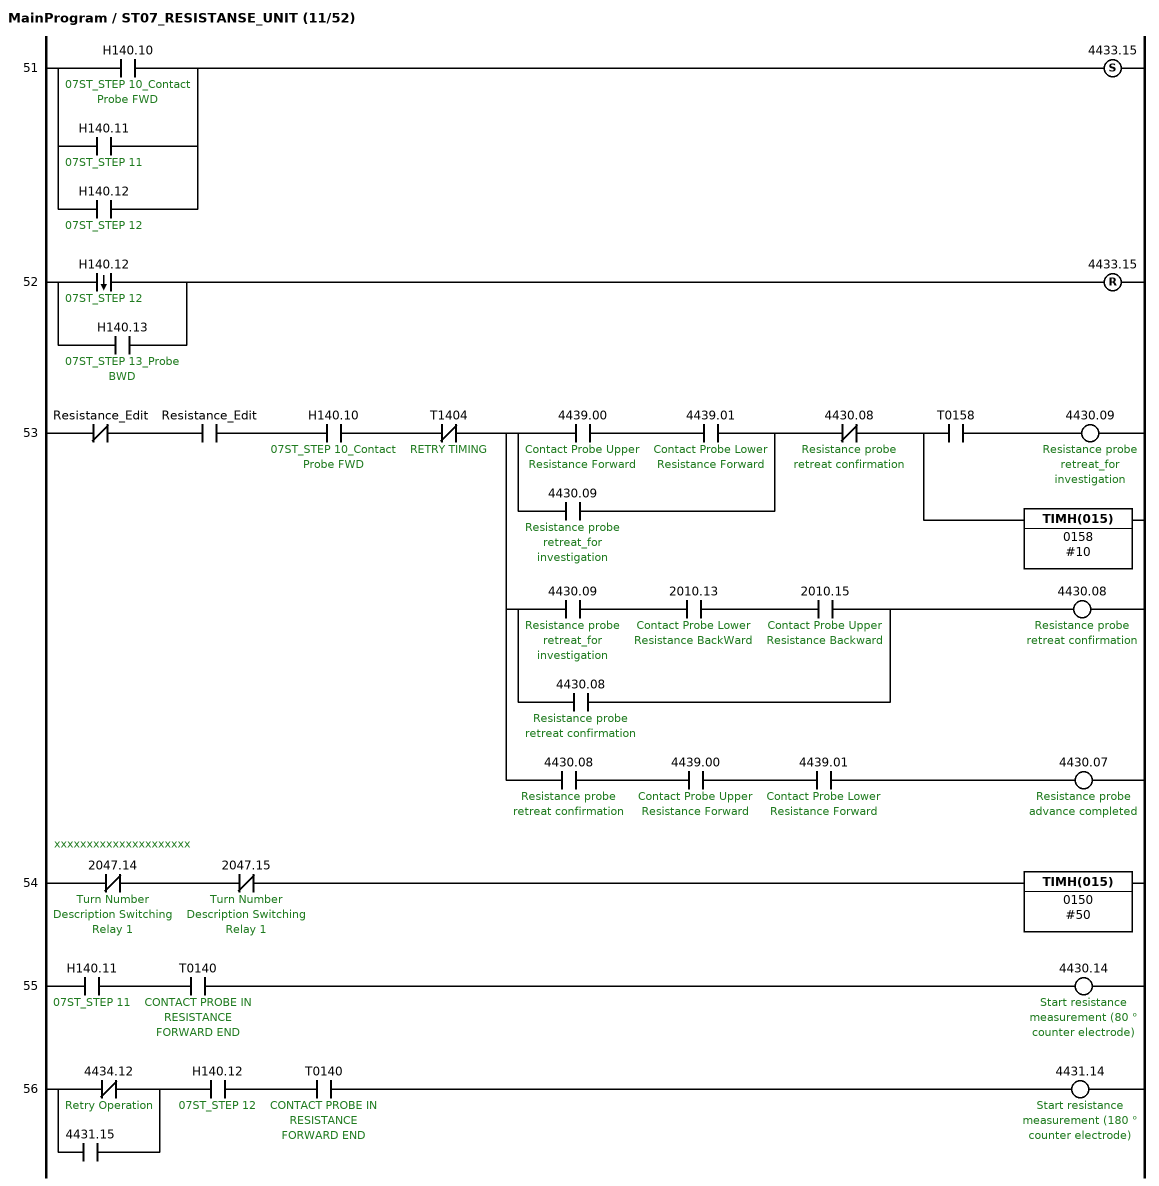
; [picture p384: MainProgram / ST07_RESISTANSE_UNIT, rungs 51-56]
; rung 51
LD H140.10  ; 07ST_STEP 10_Contact Probe FWD
OR H140.11  ; 07ST_STEP 11
OR H140.12  ; 07ST_STEP 12
SET 4433.15
; rung 52
%LD H140.12  ; 07ST_STEP 12
OR H140.13  ; 07ST_STEP 13_Probe BWD
RSET 4433.15
; rung 53
LDNOT Resistance_Edit
AND Resistance_Edit
AND H140.10  ; 07ST_STEP 10_Contact Probe FWD
ANDNOT T1404  ; RETRY TIMING
OUT TR0
LD 4439.00  ; Contact Probe Upper Resistance Forward
AND 4439.01  ; Contact Probe Lower Resistance Forward
OR 4430.09  ; Resistance probe retreat_for investigation
ANDLD
ANDNOT 4430.08  ; Resistance probe retreat confirmation
OUT TR1
AND T0158
OUT 4430.09  ; Resistance probe retreat_for investigation
LD TR1
TIMH(015) 0158 #10
LD TR0
LD 4430.09  ; Resistance probe retreat_for investigation
AND 2010.13  ; Contact Probe Lower Resistance BackWard
AND 2010.15  ; Contact Probe Upper Resistance Backward
OR 4430.08  ; Resistance probe retreat confirmation
ANDLD
OUT 4430.08  ; Resistance probe retreat confirmation
LD TR0
AND 4430.08  ; Resistance probe retreat confirmation
AND 4439.00  ; Contact Probe Upper Resistance Forward
AND 4439.01  ; Contact Probe Lower Resistance Forward
OUT 4430.07  ; Resistance probe advance completed
; rung 54: xxxxxxxxxxxxxxxxxxxxx
LDNOT 2047.14  ; Turn Number Description Switching Relay 1
ANDNOT 2047.15  ; Turn Number Description Switching Relay 1
TIMH(015) 0150 #50
; rung 55
LD H140.11  ; 07ST_STEP 11
AND T0140  ; CONTACT PROBE IN RESISTANCE FORWARD END
OUT 4430.14  ; Start resistance measurement (80 ° counter electrode)
; rung 56
LDNOT 4434.12  ; Retry Operation
OR 4431.15
AND H140.12  ; 07ST_STEP 12
AND T0140  ; CONTACT PROBE IN RESISTANCE FORWARD END
OUT 4431.14  ; Start resistance measurement (180 ° counter electrode)

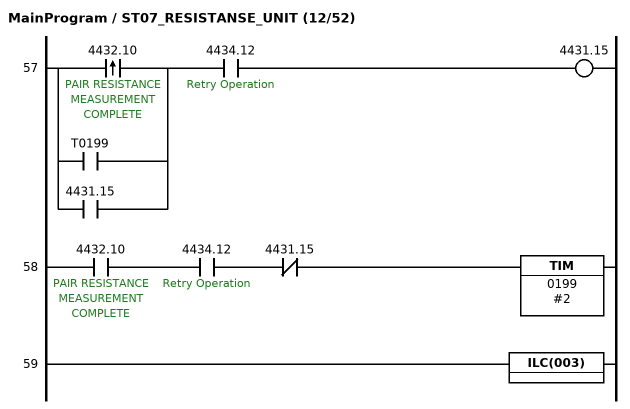
; rung 57
@LD 4432.10  ; PAIR RESISTANCE MEASUREMENT COMPLETE
OR T0199
OR 4431.15
AND 4434.12  ; Retry Operation
OUT 4431.15
; rung 58
LD 4432.10  ; PAIR RESISTANCE MEASUREMENT COMPLETE
AND 4434.12  ; Retry Operation
ANDNOT 4431.15
TIM 0199 #2
; rung 59
ILC(003)

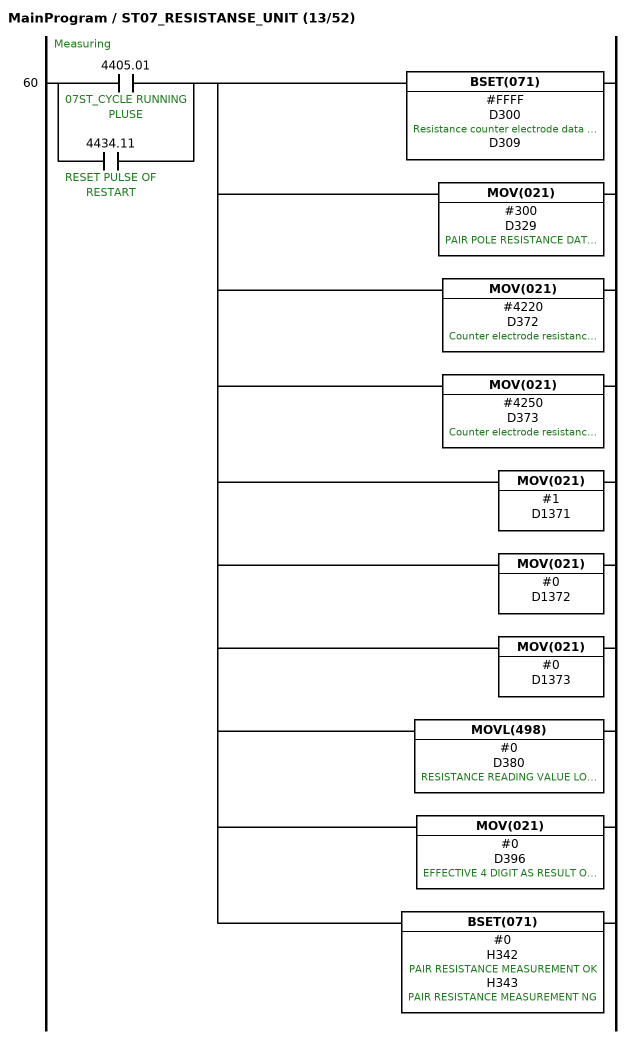
; rung 60: Measuring
LD 4405.01  ; 07ST_CYCLE RUNNING PLUSE
OR 4434.11  ; RESET PULSE OF RESTART
BSET(071) #FFFF D300 D309  ; Resistance counter electrode data 9 (80 ° counter electrode)
MOV(021) #300 D329  ; PAIR POLE RESISTANCE DATA INDIRECT SPECIFICATION
MOV(021) #4220 D372  ; Counter electrode resistance measurement indirect (80 °)
MOV(021) #4250 D373  ; Counter electrode resistance measurement indirect (80 °)
MOV(021) #1 D1371
MOV(021) #0 D1372
MOV(021) #0 D1373
MOVL(498) #0 D380  ; RESISTANCE READING VALUE LOW DIGIT
MOV(021) #0 D396  ; EFFECTIVE 4 DIGIT AS RESULT OF TEMPERATURE CORRECTION
BSET(071) #0 H342 H343  ; PAIR RESISTANCE MEASUREMENT OK, PAIR RESISTANCE MEASUREMENT NG

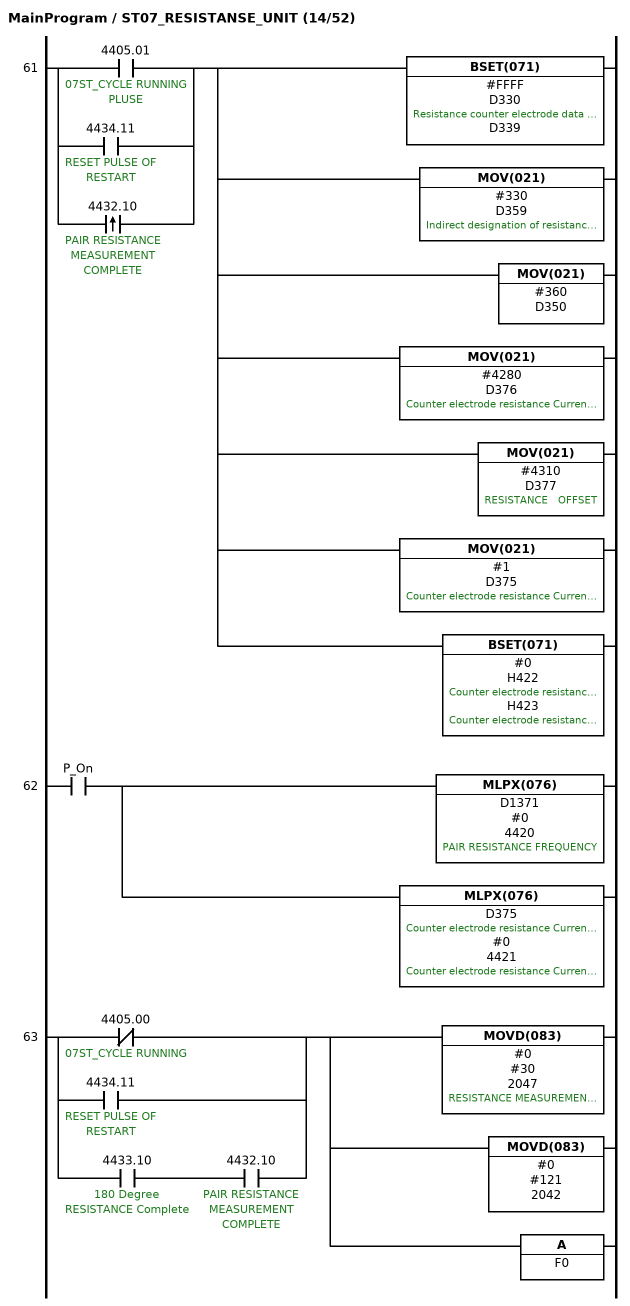
; rung 61
LD 4405.01  ; 07ST_CYCLE RUNNING PLUSE
OR 4434.11  ; RESET PULSE OF RESTART
@OR 4432.10  ; PAIR RESISTANCE MEASUREMENT COMPLETE
BSET(071) #FFFF D330 D339  ; Resistance counter electrode data 1 (180 ° counter electrode)
MOV(021) #330 D359  ; Indirect designation of resistance counter electrode data (180 °)
MOV(021) #360 D350
MOV(021) #4280 D376  ; Counter electrode resistance Current measurement count (180 °)
MOV(021) #4310 D377  ; RESISTANCE　OFFSET
MOV(021) #1 D375  ; Counter electrode resistance Current measurement count (180 °)
BSET(071) #0 H422 H423  ; Counter electrode resistance measurement OK (180 °), Counter electrode resistance measurement NG (180 °)
; rung 62
LD P_On
MLPX(076) D1371 #0 4420  ; PAIR RESISTANCE FREQUENCY
MLPX(076) D375 #0 4421  ; Counter electrode resistance Current measurement count (180 °)
; rung 63
LDNOT 4405.00  ; 07ST_CYCLE RUNNING
OR 4434.11  ; RESET PULSE OF RESTART
LD 4433.10  ; 180 Degree  RESISTANCE Complete
AND 4432.10  ; PAIR RESISTANCE MEASUREMENT COMPLETE
ORLD
MOVD(083) #0 #30 2047  ; RESISTANCE MEASUREMENT CHANGE RELAY
MOVD(083) #0 #121 2042
A  F0
// 

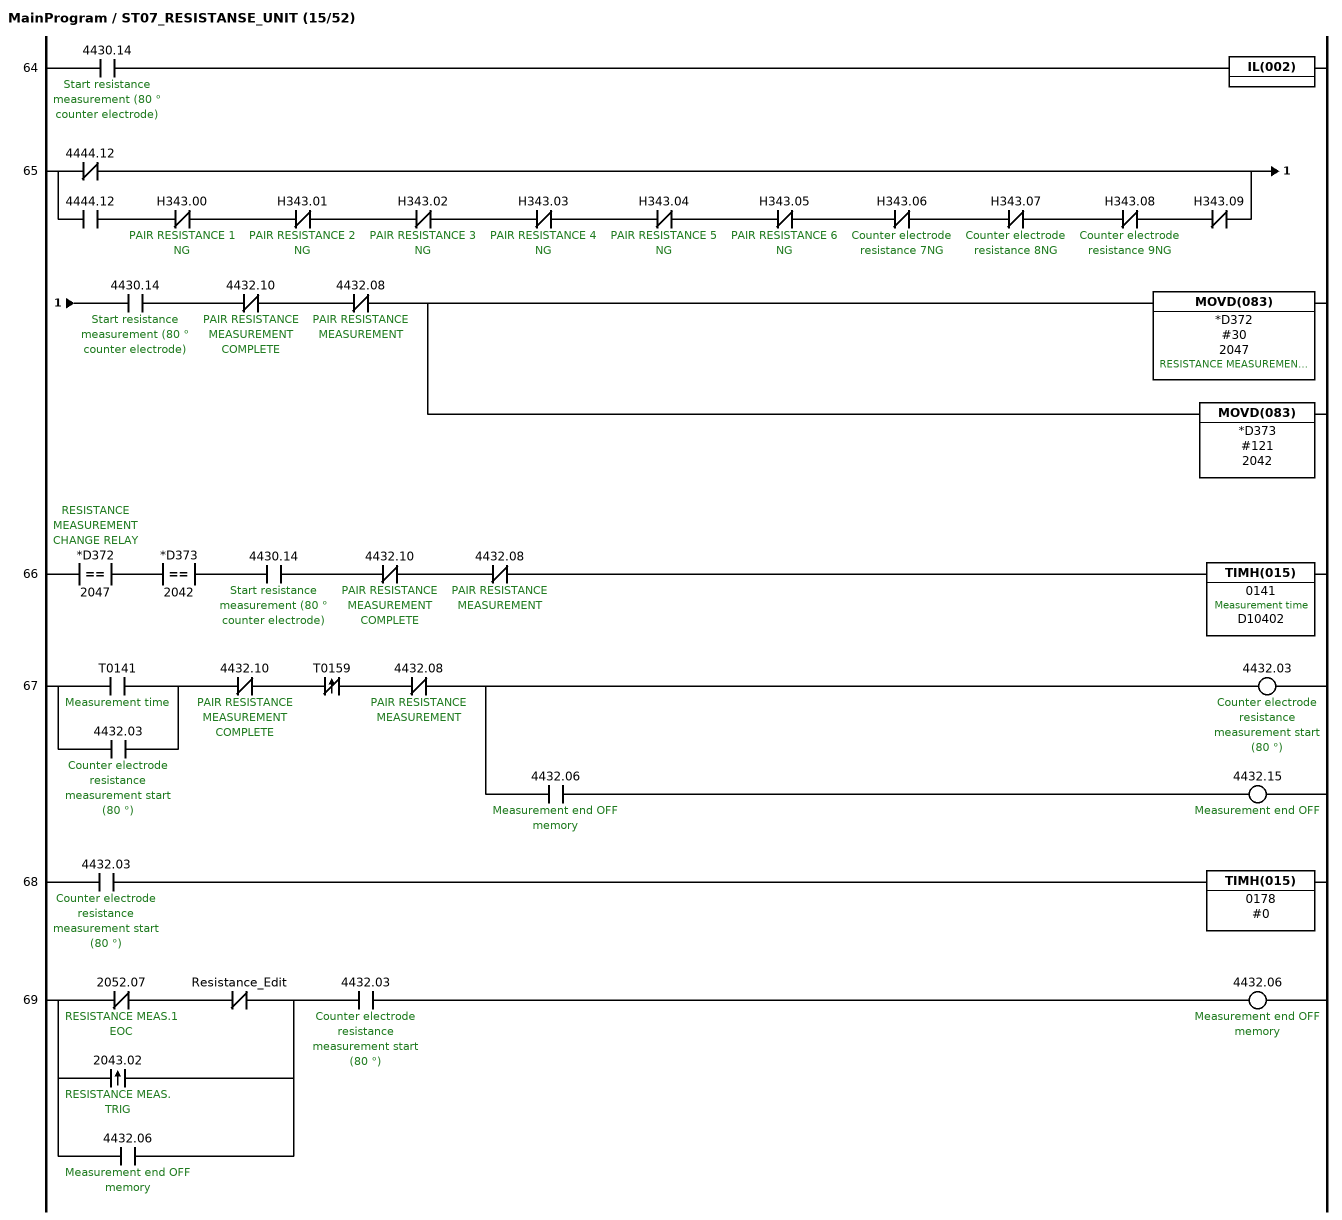
; rung 64
LD 4430.14  ; Start resistance measurement (80 ° counter electrode)
IL(002)
; rung 65
LDNOT 4444.12
LD 4444.12
ANDNOT H343.00  ; PAIR RESISTANCE 1 NG
ANDNOT H343.01  ; PAIR RESISTANCE 2 NG
ANDNOT H343.02  ; PAIR RESISTANCE 3 NG
ANDNOT H343.03  ; PAIR RESISTANCE 4 NG
ANDNOT H343.04  ; PAIR RESISTANCE 5 NG
ANDNOT H343.05  ; PAIR RESISTANCE 6 NG
ANDNOT H343.06  ; Counter electrode resistance 7NG
ANDNOT H343.07  ; Counter electrode resistance 8NG
ANDNOT H343.08  ; Counter electrode resistance 9NG
ANDNOT H343.09
ORLD
AND 4430.14  ; Start resistance measurement (80 ° counter electrode)
ANDNOT 4432.10  ; PAIR RESISTANCE MEASUREMENT COMPLETE
ANDNOT 4432.08  ; PAIR RESISTANCE MEASUREMENT
MOVD(083) *D372 #30 2047  ; RESISTANCE MEASUREMENT CHANGE RELAY
MOVD(083) *D373 #121 2042
; rung 66
LD=(300) *D372 2047  ; RESISTANCE MEASUREMENT CHANGE RELAY
AND=(300) *D373 2042
AND 4430.14  ; Start resistance measurement (80 ° counter electrode)
ANDNOT 4432.10  ; PAIR RESISTANCE MEASUREMENT COMPLETE
ANDNOT 4432.08  ; PAIR RESISTANCE MEASUREMENT
TIMH(015) 0141 D10402  ; Measurement time
; rung 67
LD T0141  ; Measurement time
OR 4432.03  ; Counter electrode resistance measurement start (80 °)
ANDNOT 4432.10  ; PAIR RESISTANCE MEASUREMENT COMPLETE
@ANDNOT T0159
ANDNOT 4432.08  ; PAIR RESISTANCE MEASUREMENT
OUT 4432.03  ; Counter electrode resistance measurement start (80 °)
AND 4432.06  ; Measurement end OFF memory
OUT 4432.15  ; Measurement end OFF
; rung 68
LD 4432.03  ; Counter electrode resistance measurement start (80 °)
TIMH(015) 0178 #0
; rung 69
LDNOT 2052.07  ; RESISTANCE MEAS.1 EOC
ANDNOT Resistance_Edit
@OR 2043.02  ; RESISTANCE MEAS. TRIG
OR 4432.06  ; Measurement end OFF memory
AND 4432.03  ; Counter electrode resistance measurement start (80 °)
OUT 4432.06  ; Measurement end OFF memory

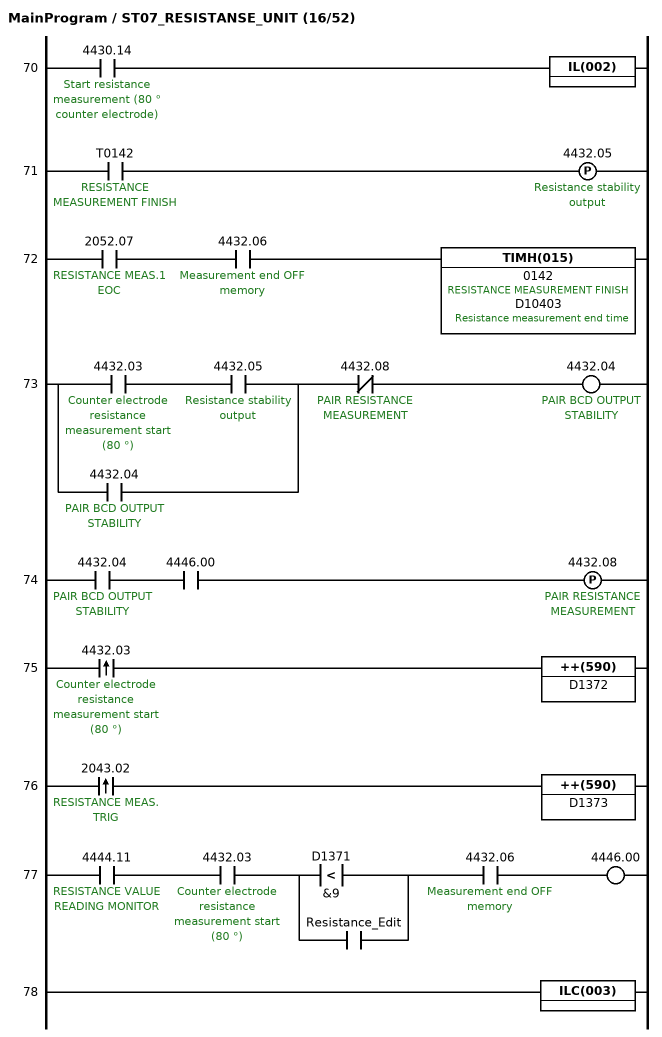
; rung 70
LD 4430.14  ; Start resistance measurement (80 ° counter electrode)
IL(002)
; rung 71
LD T0142  ; RESISTANCE MEASUREMENT FINISH
DIFU(013) 4432.05  ; Resistance stability output
; rung 72
LD 2052.07  ; RESISTANCE MEAS.1 EOC
AND 4432.06  ; Measurement end OFF memory
TIMH(015) 0142 D10403  ; Resistance measurement end time, RESISTANCE MEASUREMENT FINISH
; rung 73
LD 4432.03  ; Counter electrode resistance measurement start (80 °)
AND 4432.05  ; Resistance stability output
OR 4432.04  ; PAIR BCD OUTPUT STABILITY
ANDNOT 4432.08  ; PAIR RESISTANCE MEASUREMENT
OUT 4432.04  ; PAIR BCD OUTPUT STABILITY
; rung 74
LD 4432.04  ; PAIR BCD OUTPUT STABILITY
AND 4446.00
DIFU(013) 4432.08  ; PAIR RESISTANCE MEASUREMENT
; rung 75
@LD 4432.03  ; Counter electrode resistance measurement start (80 °)
++(590) D1372
; rung 76
@LD 2043.02  ; RESISTANCE MEAS. TRIG
++(590) D1373
; rung 77
LD 4444.11  ; RESISTANCE VALUE READING MONITOR
AND 4432.03  ; Counter electrode resistance measurement start (80 °)
LD<(310) D1371 &9
OR Resistance_Edit
ANDLD
AND 4432.06  ; Measurement end OFF memory
OUT 4446.00
; rung 78
ILC(003)

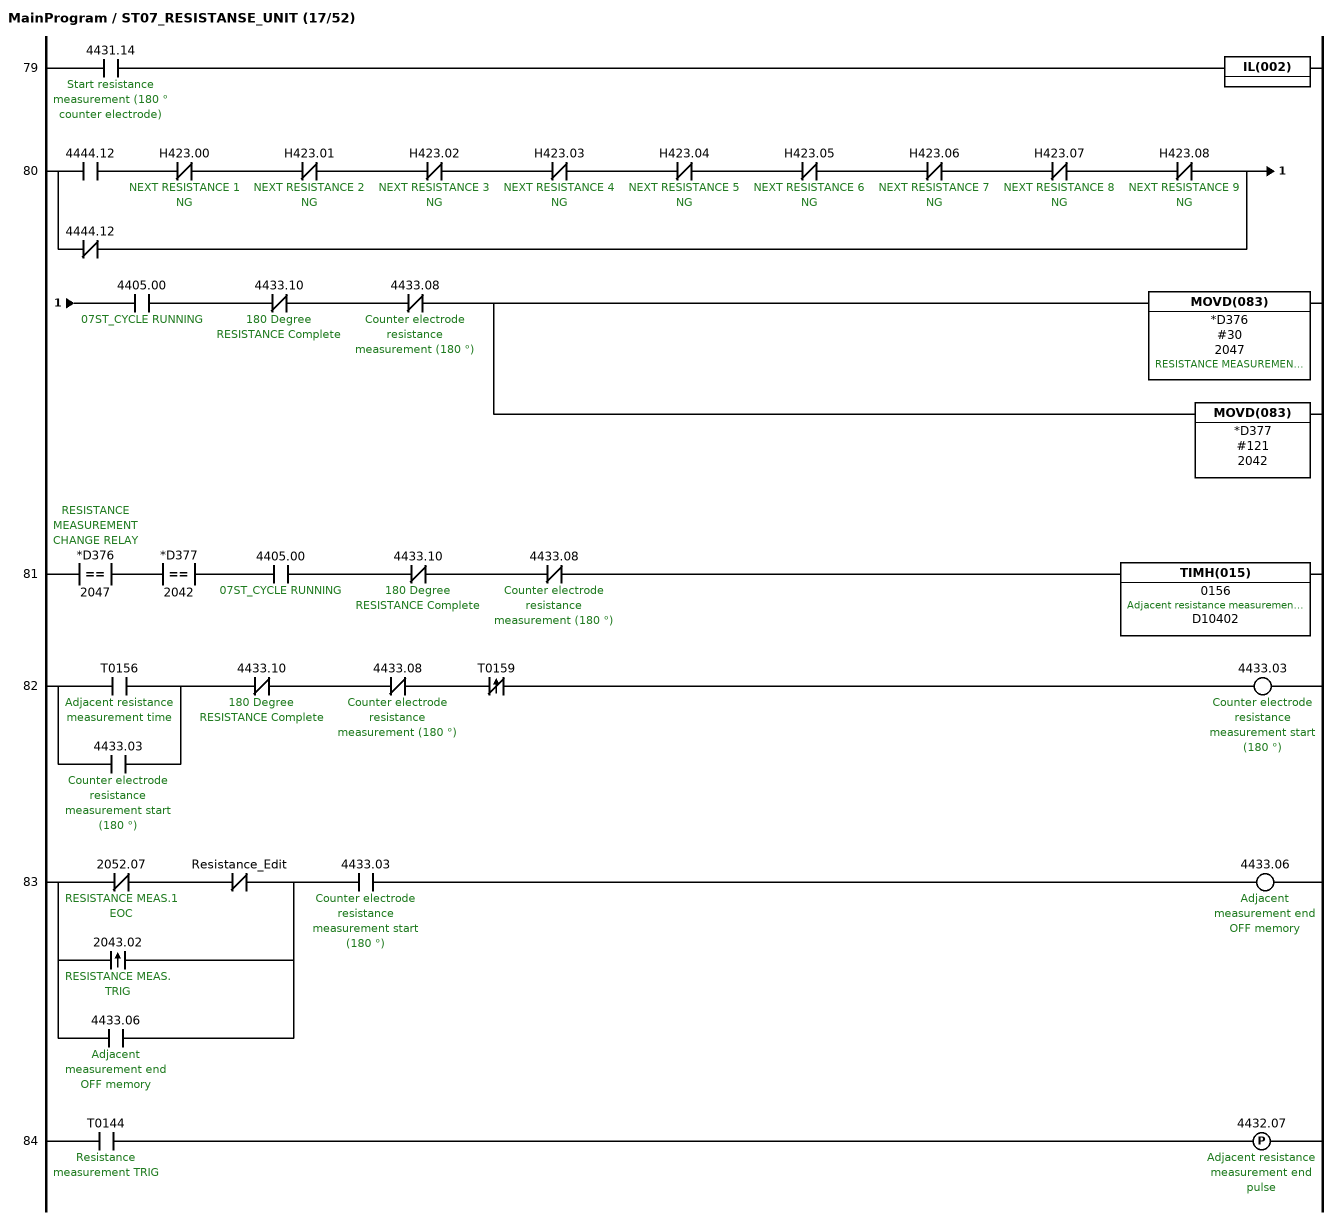
; rung 79
LD 4431.14  ; Start resistance measurement (180 ° counter electrode)
IL(002)
; rung 80
LD 4444.12
ANDNOT H423.00  ; NEXT RESISTANCE 1 NG
ANDNOT H423.01  ; NEXT RESISTANCE 2 NG
ANDNOT H423.02  ; NEXT RESISTANCE 3 NG
ANDNOT H423.03  ; NEXT RESISTANCE 4 NG
ANDNOT H423.04  ; NEXT RESISTANCE 5 NG
ANDNOT H423.05  ; NEXT RESISTANCE 6 NG
ANDNOT H423.06  ; NEXT RESISTANCE 7 NG
ANDNOT H423.07  ; NEXT RESISTANCE 8 NG
ANDNOT H423.08  ; NEXT RESISTANCE 9 NG
ORNOT 4444.12
AND 4405.00  ; 07ST_CYCLE RUNNING
ANDNOT 4433.10  ; 180 Degree  RESISTANCE Complete
ANDNOT 4433.08  ; Counter electrode resistance measurement (180 °)
MOVD(083) *D376 #30 2047  ; RESISTANCE MEASUREMENT CHANGE RELAY
MOVD(083) *D377 #121 2042
; rung 81
LD=(300) *D376 2047  ; RESISTANCE MEASUREMENT CHANGE RELAY
AND=(300) *D377 2042
AND 4405.00  ; 07ST_CYCLE RUNNING
ANDNOT 4433.10  ; 180 Degree  RESISTANCE Complete
ANDNOT 4433.08  ; Counter electrode resistance measurement (180 °)
TIMH(015) 0156 D10402  ; Adjacent resistance measurement time
; rung 82
LD T0156  ; Adjacent resistance measurement time
OR 4433.03  ; Counter electrode resistance measurement start (180 °)
ANDNOT 4433.10  ; 180 Degree  RESISTANCE Complete
ANDNOT 4433.08  ; Counter electrode resistance measurement (180 °)
@ANDNOT T0159
OUT 4433.03  ; Counter electrode resistance measurement start (180 °)
; rung 83
LDNOT 2052.07  ; RESISTANCE MEAS.1 EOC
ANDNOT Resistance_Edit
@OR 2043.02  ; RESISTANCE MEAS. TRIG
OR 4433.06  ; Adjacent measurement end OFF memory
AND 4433.03  ; Counter electrode resistance measurement start (180 °)
OUT 4433.06  ; Adjacent measurement end OFF memory
; rung 84
LD T0144  ; Resistance measurement TRIG
DIFU(013) 4432.07  ; Adjacent resistance measurement end pulse

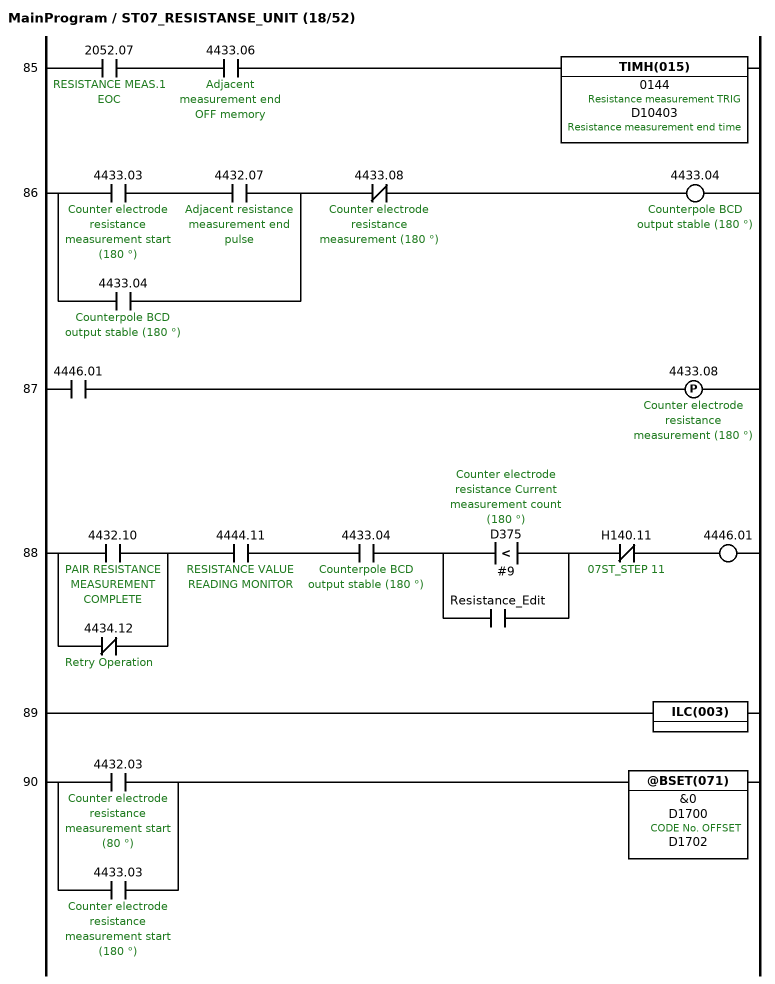
; rung 85
LD 2052.07  ; RESISTANCE MEAS.1 EOC
AND 4433.06  ; Adjacent measurement end OFF memory
TIMH(015) 0144 D10403  ; Resistance measurement end time, Resistance measurement TRIG
; rung 86
LD 4433.03  ; Counter electrode resistance measurement start (180 °)
AND 4432.07  ; Adjacent resistance measurement end pulse
OR 4433.04  ; Counterpole BCD output stable (180 °)
ANDNOT 4433.08  ; Counter electrode resistance measurement (180 °)
OUT 4433.04  ; Counterpole BCD output stable (180 °)
; rung 87
LD 4446.01
DIFU(013) 4433.08  ; Counter electrode resistance measurement (180 °)
; rung 88
LD 4432.10  ; PAIR RESISTANCE MEASUREMENT COMPLETE
ORNOT 4434.12  ; Retry Operation
AND 4444.11  ; RESISTANCE VALUE READING MONITOR
AND 4433.04  ; Counterpole BCD output stable (180 °)
LD<(310) D375 #9  ; Counter electrode resistance Current measurement count (180 °)
OR Resistance_Edit
ANDLD
ANDNOT H140.11  ; 07ST_STEP 11
OUT 4446.01
; rung 89
ILC(003)
; rung 90
LD 4432.03  ; Counter electrode resistance measurement start (80 °)
OR 4433.03  ; Counter electrode resistance measurement start (180 °)
@BSET(071) &0 D1700 D1702  ; CODE No. OFFSET

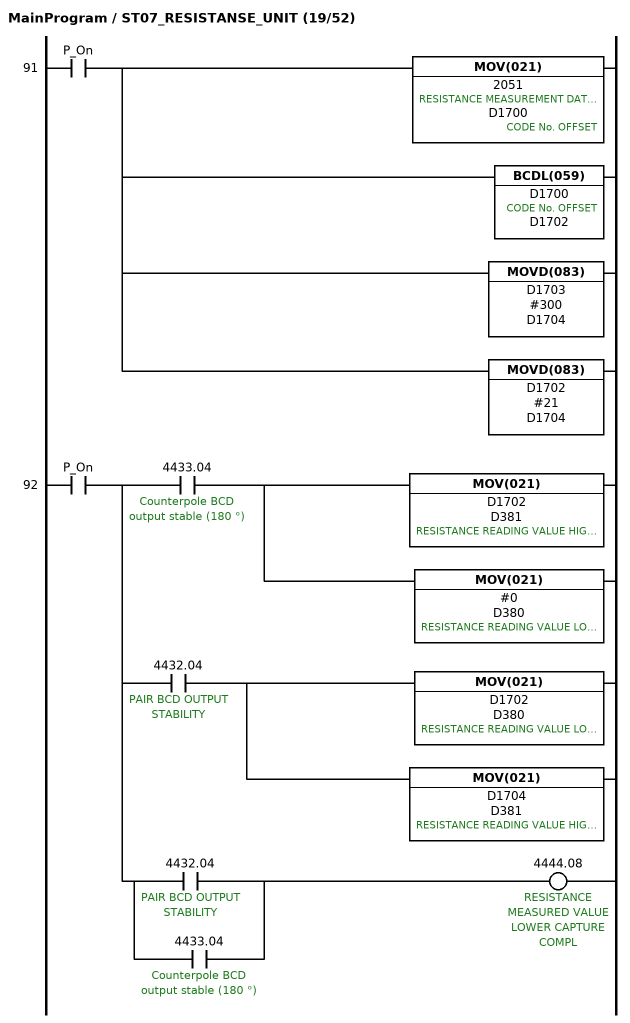
; rung 91
LD P_On
MOV(021) 2051 D1700  ; RESISTANCE MEASUREMENT DATA BCD, CODE No. OFFSET
BCDL(059) D1700 D1702  ; CODE No. OFFSET
MOVD(083) D1703 #300 D1704
MOVD(083) D1702 #21 D1704
; rung 92
LD P_On
OUT TR0
AND 4433.04  ; Counterpole BCD output stable (180 °)
MOV(021) D1702 D381  ; RESISTANCE READING VALUE HIGH DIGIT
MOV(021) #0 D380  ; RESISTANCE READING VALUE LOW DIGIT
LD TR0
AND 4432.04  ; PAIR BCD OUTPUT STABILITY
MOV(021) D1702 D380  ; RESISTANCE READING VALUE LOW DIGIT
MOV(021) D1704 D381  ; RESISTANCE READING VALUE HIGH DIGIT
LD TR0
LD 4432.04  ; PAIR BCD OUTPUT STABILITY
OR 4433.04  ; Counterpole BCD output stable (180 °)
ANDLD
OUT 4444.08  ; RESISTANCE MEASURED VALUE LOWER CAPTURE COMPL

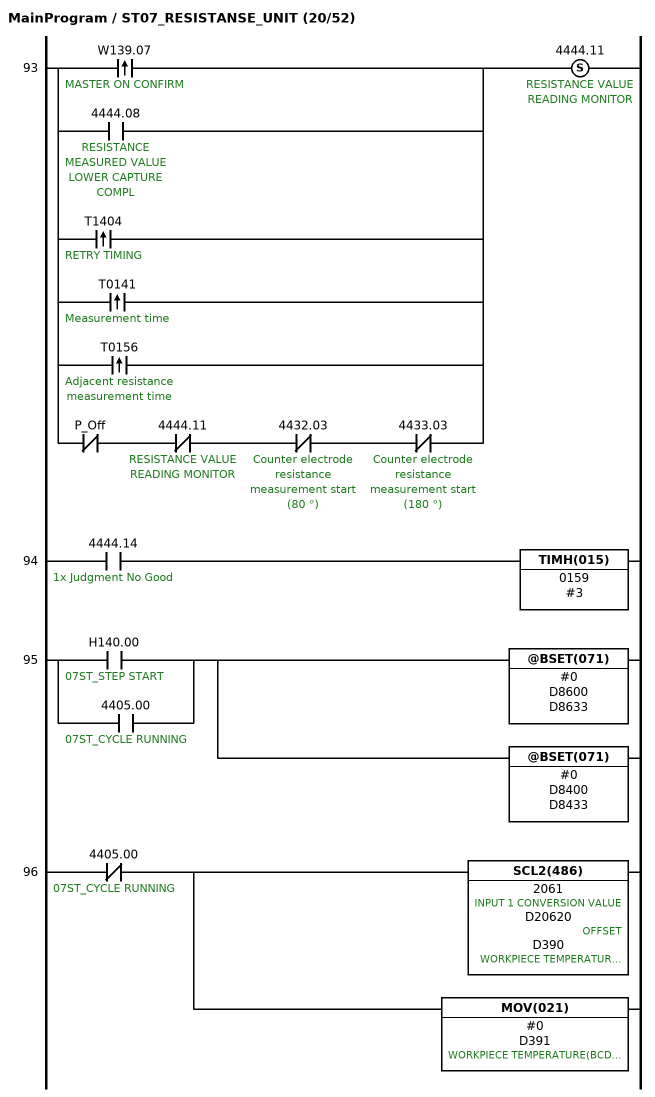
; rung 93
@LD W139.07  ; MASTER ON CONFIRM
OR 4444.08  ; RESISTANCE MEASURED VALUE LOWER CAPTURE COMPL
@OR T1404  ; RETRY TIMING
@OR T0141  ; Measurement time
@OR T0156  ; Adjacent resistance measurement time
LDNOT P_Off
ANDNOT 4444.11  ; RESISTANCE VALUE READING MONITOR
ANDNOT 4432.03  ; Counter electrode resistance measurement start (80 °)
ANDNOT 4433.03  ; Counter electrode resistance measurement start (180 °)
ORLD
SET 4444.11  ; RESISTANCE VALUE READING MONITOR
; rung 94
LD 4444.14  ; 1x Judgment No Good
TIMH(015) 0159 #3
; rung 95
LD H140.00  ; 07ST_STEP START
OR 4405.00  ; 07ST_CYCLE RUNNING
@BSET(071) #0 D8600 D8633
@BSET(071) #0 D8400 D8433
; rung 96
LDNOT 4405.00  ; 07ST_CYCLE RUNNING
SCL2(486) 2061 D20620 D390  ; INPUT 1 CONVERSION VALUE, OFFSET, WORKPIECE TEMPERATURE READING(BCD)  // The scaled temperature is forwarded
MOV(021) #0 D391  ; WORKPIECE TEMPERATURE(BCD) HIGH DIGIT

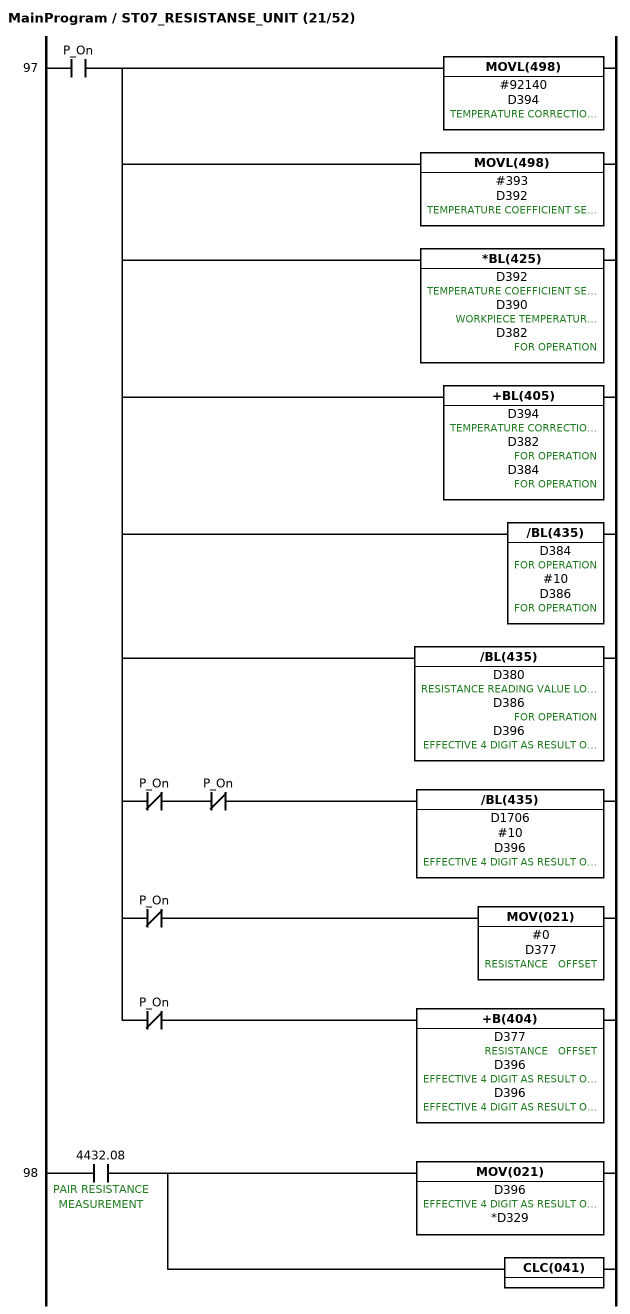
; rung 97
LD P_On
OUT TR0
MOVL(498) #92140 D394  ; TEMPERATURE CORRECTION OPERATION LOW DIGIT
MOVL(498) #393 D392  ; TEMPERATURE COEFFICIENT SET VALUE
*BL(425) D392 D390 D382  ; TEMPERATURE COEFFICIENT SET VALUE, WORKPIECE TEMPERATURE READING(BCD), FOR OPERATION
+BL(405) D394 D382 D384  ; TEMPERATURE CORRECTION OPERATION LOW DIGIT, FOR OPERATION
/BL(435) D384 #10 D386  ; FOR OPERATION
/BL(435) D380 D386 D396  ; RESISTANCE READING VALUE LOW DIGIT, FOR OPERATION, EFFECTIVE 4 DIGIT AS RESULT OF TEMPERATURE CORRECTION
ANDNOT P_On
ANDNOT P_On
/BL(435) D1706 #10 D396  ; EFFECTIVE 4 DIGIT AS RESULT OF TEMPERATURE CORRECTION
LD TR0
ANDNOT P_On
MOV(021) #0 D377  ; RESISTANCE　OFFSET
LD TR0
ANDNOT P_On
+B(404) D377 D396 D396  ; RESISTANCE　OFFSET, EFFECTIVE 4 DIGIT AS RESULT OF TEMPERATURE CORRECTION
; rung 98
LD 4432.08  ; PAIR RESISTANCE MEASUREMENT
MOV(021) D396 *D329  ; EFFECTIVE 4 DIGIT AS RESULT OF TEMPERATURE CORRECTION  // The data that has been corrected is transmitted
CLC(041)

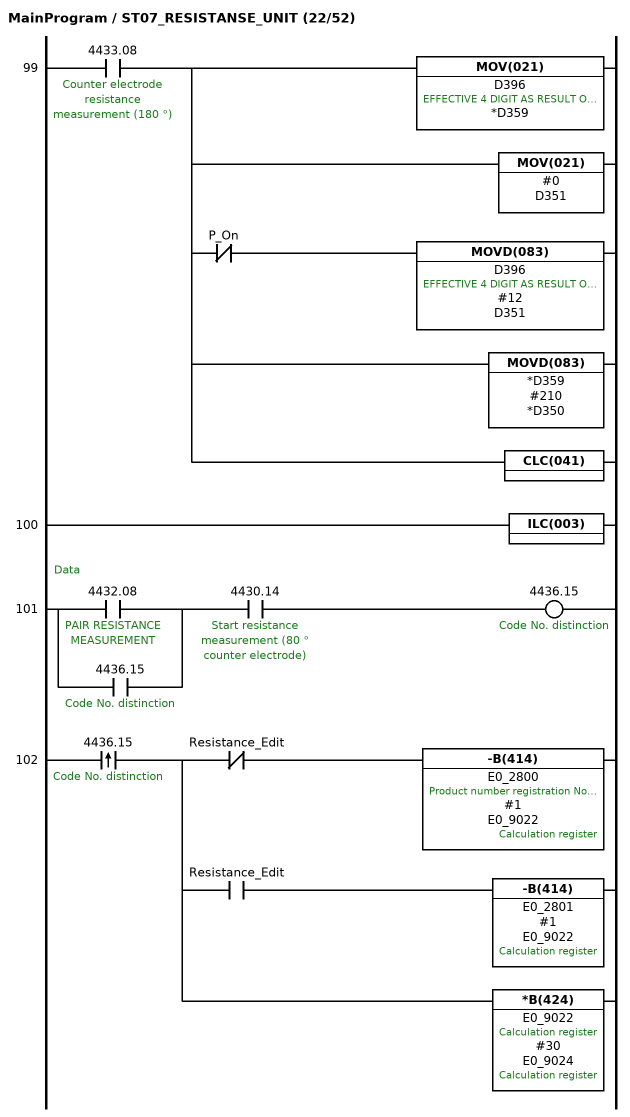
; rung 99
LD 4433.08  ; Counter electrode resistance measurement (180 °)
OUT TR0
MOV(021) D396 *D359  ; EFFECTIVE 4 DIGIT AS RESULT OF TEMPERATURE CORRECTION
MOV(021) #0 D351
ANDNOT P_On
MOVD(083) D396 #12 D351  ; EFFECTIVE 4 DIGIT AS RESULT OF TEMPERATURE CORRECTION
LD TR0
MOVD(083) *D359 #210 *D350
CLC(041)
; rung 100
ILC(003)
; rung 101: Data
LD 4432.08  ; PAIR RESISTANCE MEASUREMENT
OR 4436.15  ; Code No. distinction
AND 4430.14  ; Start resistance measurement (80 ° counter electrode)
OUT 4436.15  ; Code No. distinction
; rung 102
@LD 4436.15  ; Code No. distinction
OUT TR0
ANDNOT Resistance_Edit
-B(414) E0_2800 #1 E0_9022  ; Product number registration No. (resistance measurement ST), Calculation register
LD TR0
AND Resistance_Edit
-B(414) E0_2801 #1 E0_9022  ; Calculation register
LD TR0
*B(424) E0_9022 #30 E0_9024  ; Calculation register

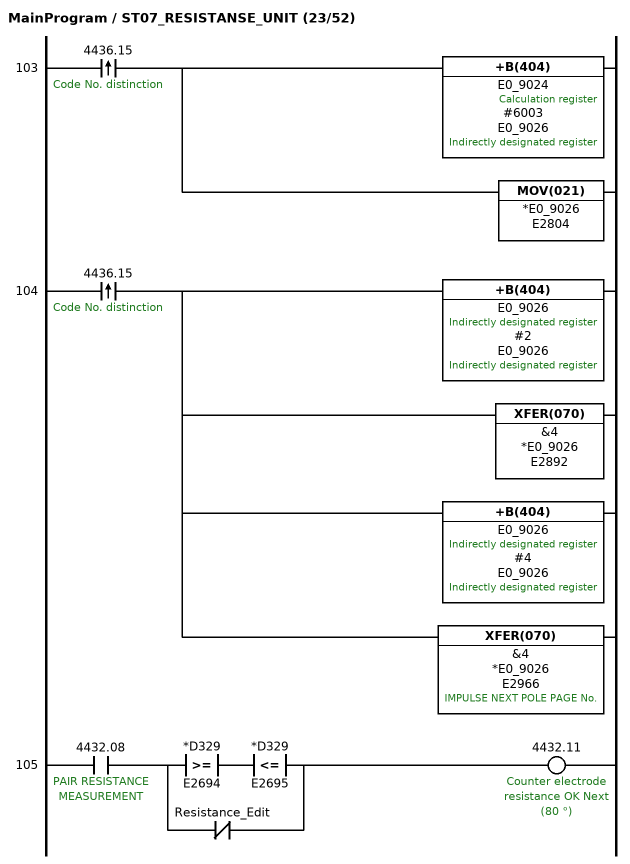
; rung 103
@LD 4436.15  ; Code No. distinction
+B(404) E0_9024 #6003 E0_9026  ; Calculation register, Indirectly designated register
MOV(021) *E0_9026 E2804
; rung 104
@LD 4436.15  ; Code No. distinction
+B(404) E0_9026 #2 E0_9026  ; Indirectly designated register
XFER(070) &4 *E0_9026 E2892
+B(404) E0_9026 #4 E0_9026  ; Indirectly designated register
XFER(070) &4 *E0_9026 E2966  ; IMPULSE NEXT POLE PAGE No.
; rung 105
LD 4432.08  ; PAIR RESISTANCE MEASUREMENT
LD>=(325) *D329 E2694
AND<=(315) *D329 E2695
ORNOT Resistance_Edit
ANDLD
OUT 4432.11  ; Counter electrode resistance OK Next (80 °)

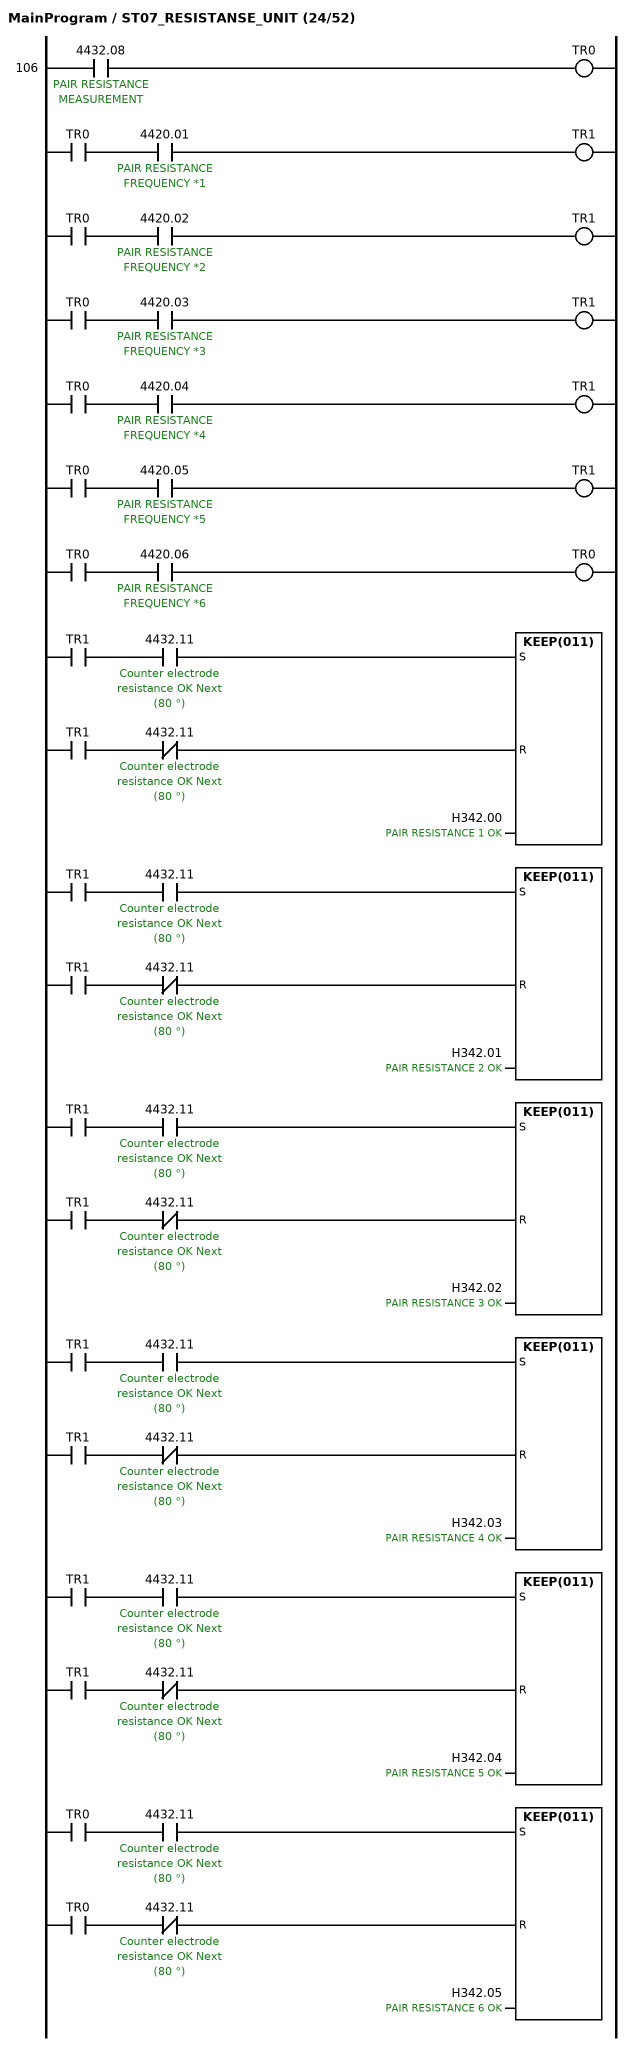
; rung 106
LD 4432.08  ; PAIR RESISTANCE MEASUREMENT
OUT TR0
AND 4420.01  ; PAIR RESISTANCE FREQUENCY *1
OUT TR1
AND 4432.11  ; Counter electrode resistance OK Next (80 °)
LD TR1
ANDNOT 4432.11  ; Counter electrode resistance OK Next (80 °)
KEEP(011) H342.00  ; PAIR RESISTANCE 1 OK
LD TR0
AND 4420.02  ; PAIR RESISTANCE FREQUENCY *2
OUT TR1
AND 4432.11  ; Counter electrode resistance OK Next (80 °)
LD TR1
ANDNOT 4432.11  ; Counter electrode resistance OK Next (80 °)
KEEP(011) H342.01  ; PAIR RESISTANCE 2 OK
LD TR0
AND 4420.03  ; PAIR RESISTANCE FREQUENCY *3
OUT TR1
AND 4432.11  ; Counter electrode resistance OK Next (80 °)
LD TR1
ANDNOT 4432.11  ; Counter electrode resistance OK Next (80 °)
KEEP(011) H342.02  ; PAIR RESISTANCE 3 OK
LD TR0
AND 4420.04  ; PAIR RESISTANCE FREQUENCY *4
OUT TR1
AND 4432.11  ; Counter electrode resistance OK Next (80 °)
LD TR1
ANDNOT 4432.11  ; Counter electrode resistance OK Next (80 °)
KEEP(011) H342.03  ; PAIR RESISTANCE 4 OK
LD TR0
AND 4420.05  ; PAIR RESISTANCE FREQUENCY *5
OUT TR1
AND 4432.11  ; Counter electrode resistance OK Next (80 °)
LD TR1
ANDNOT 4432.11  ; Counter electrode resistance OK Next (80 °)
KEEP(011) H342.04  ; PAIR RESISTANCE 5 OK
LD TR0
AND 4420.06  ; PAIR RESISTANCE FREQUENCY *6
OUT TR0
AND 4432.11  ; Counter electrode resistance OK Next (80 °)
LD TR0
ANDNOT 4432.11  ; Counter electrode resistance OK Next (80 °)
KEEP(011) H342.05  ; PAIR RESISTANCE 6 OK

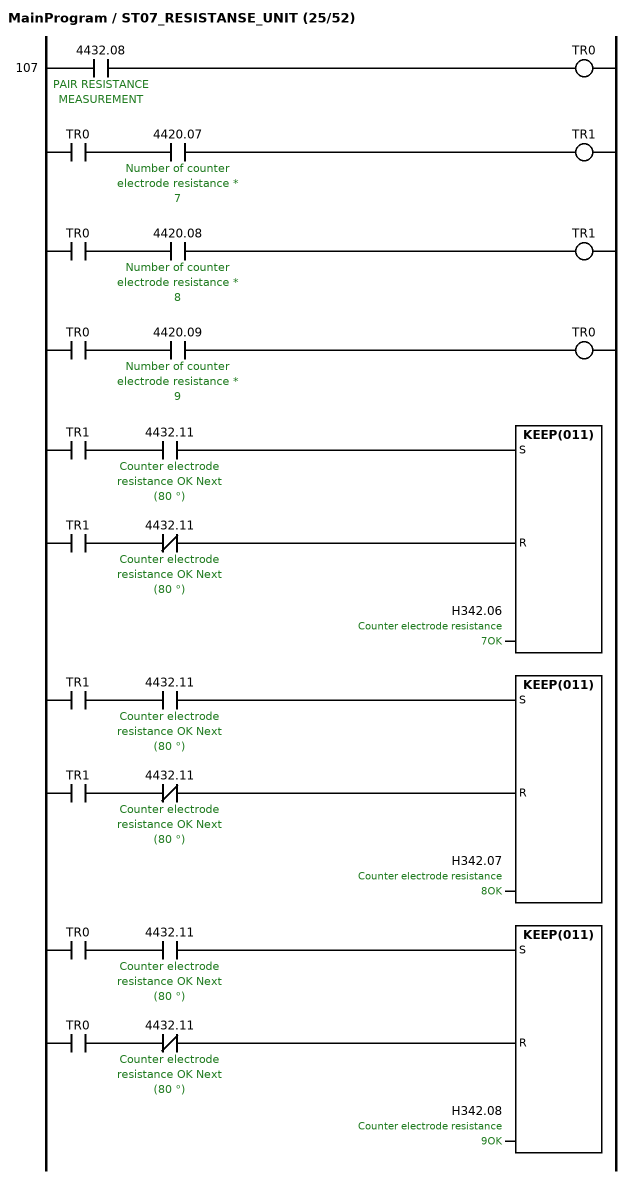
; rung 107
LD 4432.08  ; PAIR RESISTANCE MEASUREMENT
OUT TR0
AND 4420.07  ; Number of counter electrode resistance * 7
OUT TR1
AND 4432.11  ; Counter electrode resistance OK Next (80 °)
LD TR1
ANDNOT 4432.11  ; Counter electrode resistance OK Next (80 °)
KEEP(011) H342.06  ; Counter electrode resistance 7OK
LD TR0
AND 4420.08  ; Number of counter electrode resistance * 8
OUT TR1
AND 4432.11  ; Counter electrode resistance OK Next (80 °)
LD TR1
ANDNOT 4432.11  ; Counter electrode resistance OK Next (80 °)
KEEP(011) H342.07  ; Counter electrode resistance 8OK
LD TR0
AND 4420.09  ; Number of counter electrode resistance * 9
OUT TR0
AND 4432.11  ; Counter electrode resistance OK Next (80 °)
LD TR0
ANDNOT 4432.11  ; Counter electrode resistance OK Next (80 °)
KEEP(011) H342.08  ; Counter electrode resistance 9OK

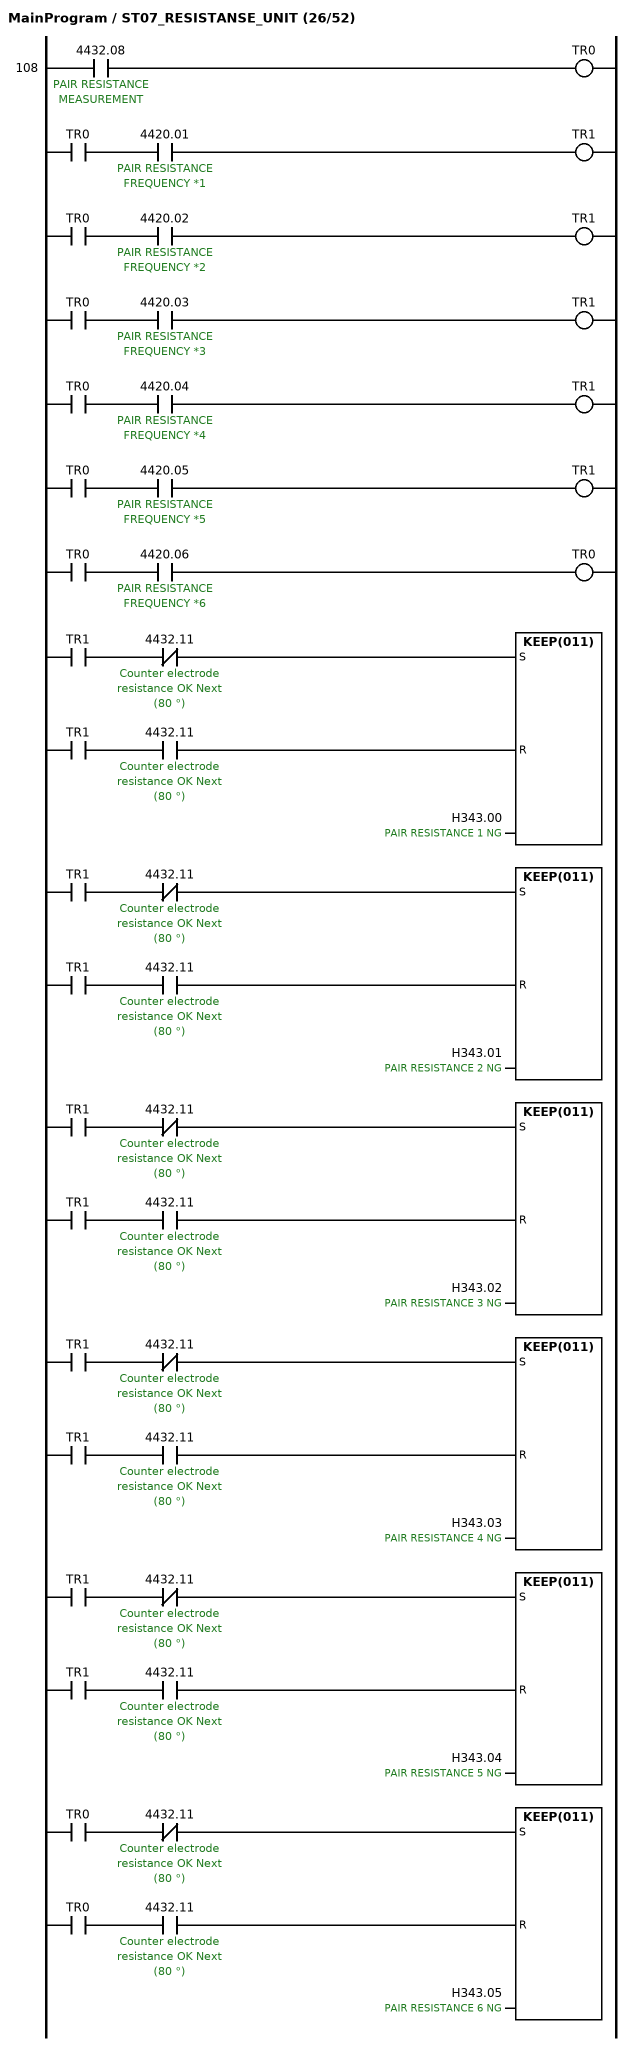
; rung 108
LD 4432.08  ; PAIR RESISTANCE MEASUREMENT
OUT TR0
AND 4420.01  ; PAIR RESISTANCE FREQUENCY *1
OUT TR1
ANDNOT 4432.11  ; Counter electrode resistance OK Next (80 °)
LD TR1
AND 4432.11  ; Counter electrode resistance OK Next (80 °)
KEEP(011) H343.00  ; PAIR RESISTANCE 1 NG
LD TR0
AND 4420.02  ; PAIR RESISTANCE FREQUENCY *2
OUT TR1
ANDNOT 4432.11  ; Counter electrode resistance OK Next (80 °)
LD TR1
AND 4432.11  ; Counter electrode resistance OK Next (80 °)
KEEP(011) H343.01  ; PAIR RESISTANCE 2 NG
LD TR0
AND 4420.03  ; PAIR RESISTANCE FREQUENCY *3
OUT TR1
ANDNOT 4432.11  ; Counter electrode resistance OK Next (80 °)
LD TR1
AND 4432.11  ; Counter electrode resistance OK Next (80 °)
KEEP(011) H343.02  ; PAIR RESISTANCE 3 NG
LD TR0
AND 4420.04  ; PAIR RESISTANCE FREQUENCY *4
OUT TR1
ANDNOT 4432.11  ; Counter electrode resistance OK Next (80 °)
LD TR1
AND 4432.11  ; Counter electrode resistance OK Next (80 °)
KEEP(011) H343.03  ; PAIR RESISTANCE 4 NG
LD TR0
AND 4420.05  ; PAIR RESISTANCE FREQUENCY *5
OUT TR1
ANDNOT 4432.11  ; Counter electrode resistance OK Next (80 °)
LD TR1
AND 4432.11  ; Counter electrode resistance OK Next (80 °)
KEEP(011) H343.04  ; PAIR RESISTANCE 5 NG
LD TR0
AND 4420.06  ; PAIR RESISTANCE FREQUENCY *6
OUT TR0
ANDNOT 4432.11  ; Counter electrode resistance OK Next (80 °)
LD TR0
AND 4432.11  ; Counter electrode resistance OK Next (80 °)
KEEP(011) H343.05  ; PAIR RESISTANCE 6 NG

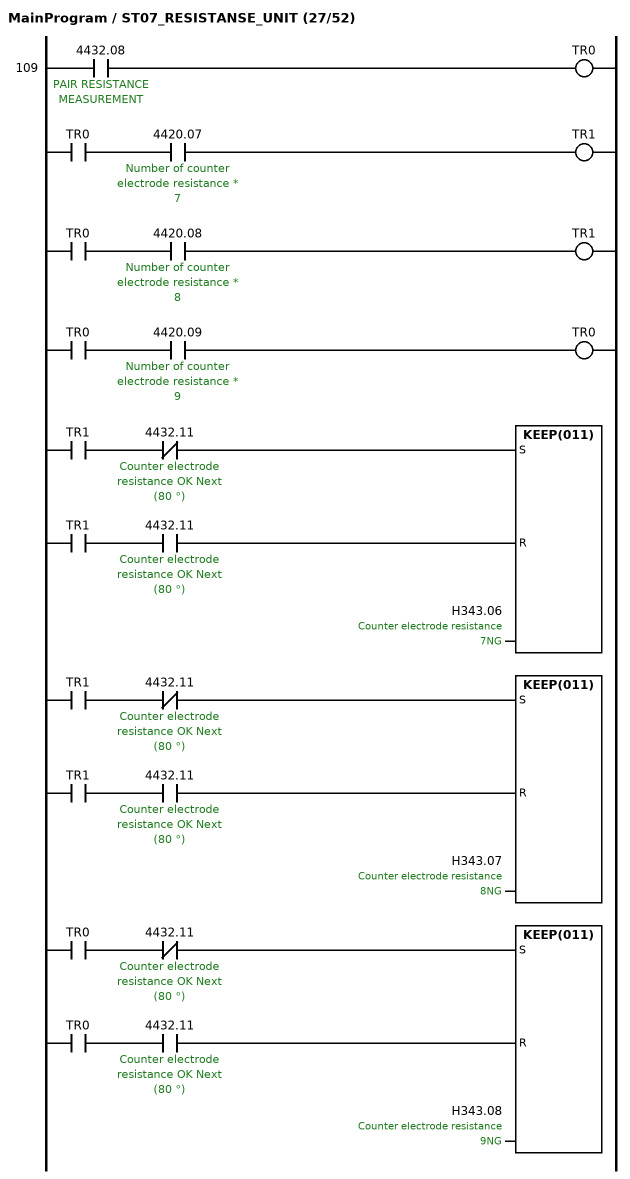
; rung 109
LD 4432.08  ; PAIR RESISTANCE MEASUREMENT
OUT TR0
AND 4420.07  ; Number of counter electrode resistance * 7
OUT TR1
ANDNOT 4432.11  ; Counter electrode resistance OK Next (80 °)
LD TR1
AND 4432.11  ; Counter electrode resistance OK Next (80 °)
KEEP(011) H343.06  ; Counter electrode resistance 7NG
LD TR0
AND 4420.08  ; Number of counter electrode resistance * 8
OUT TR1
ANDNOT 4432.11  ; Counter electrode resistance OK Next (80 °)
LD TR1
AND 4432.11  ; Counter electrode resistance OK Next (80 °)
KEEP(011) H343.07  ; Counter electrode resistance 8NG
LD TR0
AND 4420.09  ; Number of counter electrode resistance * 9
OUT TR0
ANDNOT 4432.11  ; Counter electrode resistance OK Next (80 °)
LD TR0
AND 4432.11  ; Counter electrode resistance OK Next (80 °)
KEEP(011) H343.08  ; Counter electrode resistance 9NG

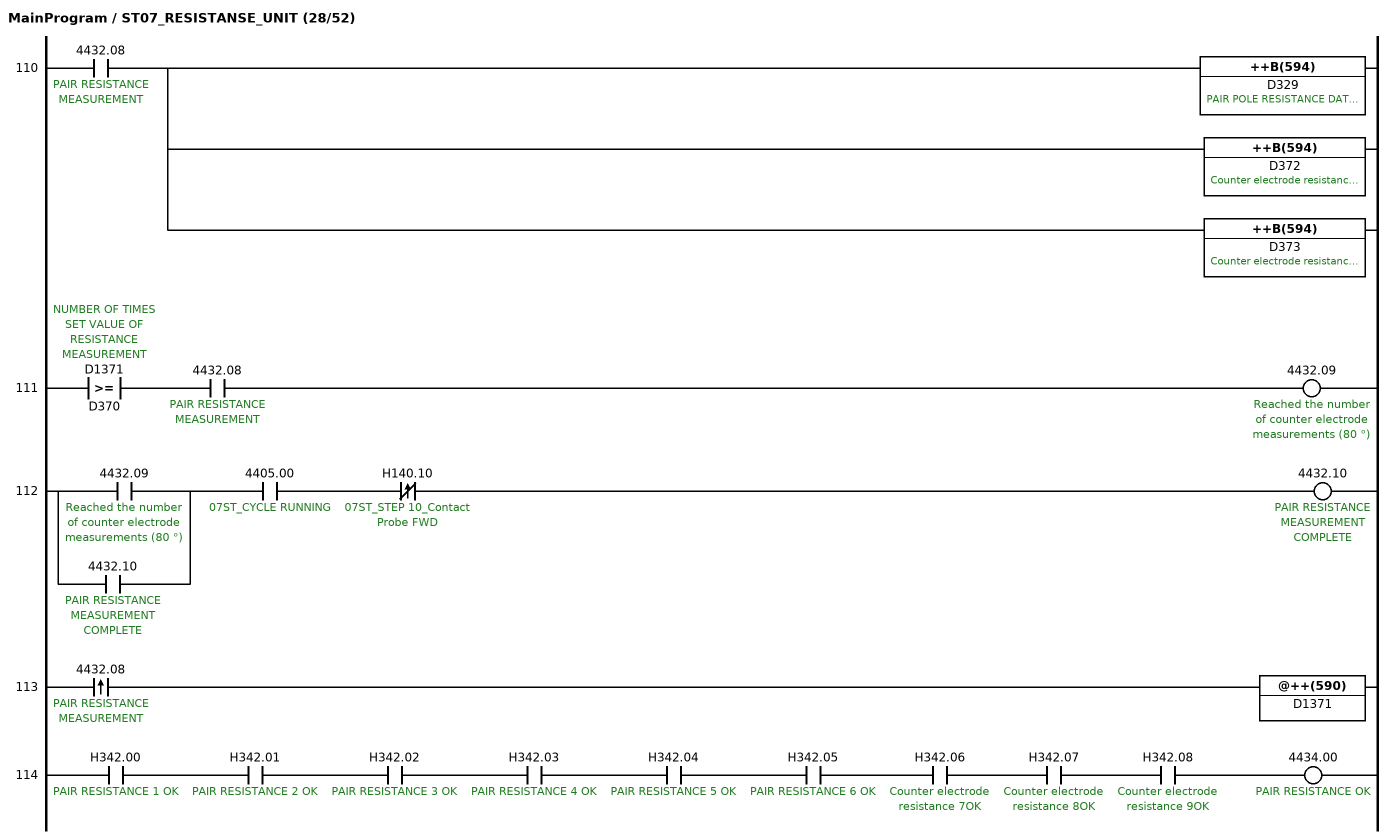
; rung 110
LD 4432.08  ; PAIR RESISTANCE MEASUREMENT
++B(594) D329  ; PAIR POLE RESISTANCE DATA INDIRECT SPECIFICATION
++B(594) D372  ; Counter electrode resistance measurement indirect (80 °)
++B(594) D373  ; Counter electrode resistance measurement indirect (80 °)  // 
; rung 111
LD>=(325) D1371 D370  ; NUMBER OF TIMES SET VALUE OF RESISTANCE MEASUREMENT
AND 4432.08  ; PAIR RESISTANCE MEASUREMENT
OUT 4432.09  ; Reached the number of counter electrode measurements (80 °)
; rung 112
LD 4432.09  ; Reached the number of counter electrode measurements (80 °)
OR 4432.10  ; PAIR RESISTANCE MEASUREMENT COMPLETE
AND 4405.00  ; 07ST_CYCLE RUNNING
@ANDNOT H140.10  ; 07ST_STEP 10_Contact Probe FWD
OUT 4432.10  ; PAIR RESISTANCE MEASUREMENT COMPLETE
; rung 113
@LD 4432.08  ; PAIR RESISTANCE MEASUREMENT
@++(590) D1371
; rung 114
LD H342.00  ; PAIR RESISTANCE 1 OK
AND H342.01  ; PAIR RESISTANCE 2 OK
AND H342.02  ; PAIR RESISTANCE 3 OK
AND H342.03  ; PAIR RESISTANCE 4 OK
AND H342.04  ; PAIR RESISTANCE 5 OK
AND H342.05  ; PAIR RESISTANCE 6 OK
AND H342.06  ; Counter electrode resistance 7OK
AND H342.07  ; Counter electrode resistance 8OK
AND H342.08  ; Counter electrode resistance 9OK
OUT 4434.00  ; PAIR RESISTANCE OK

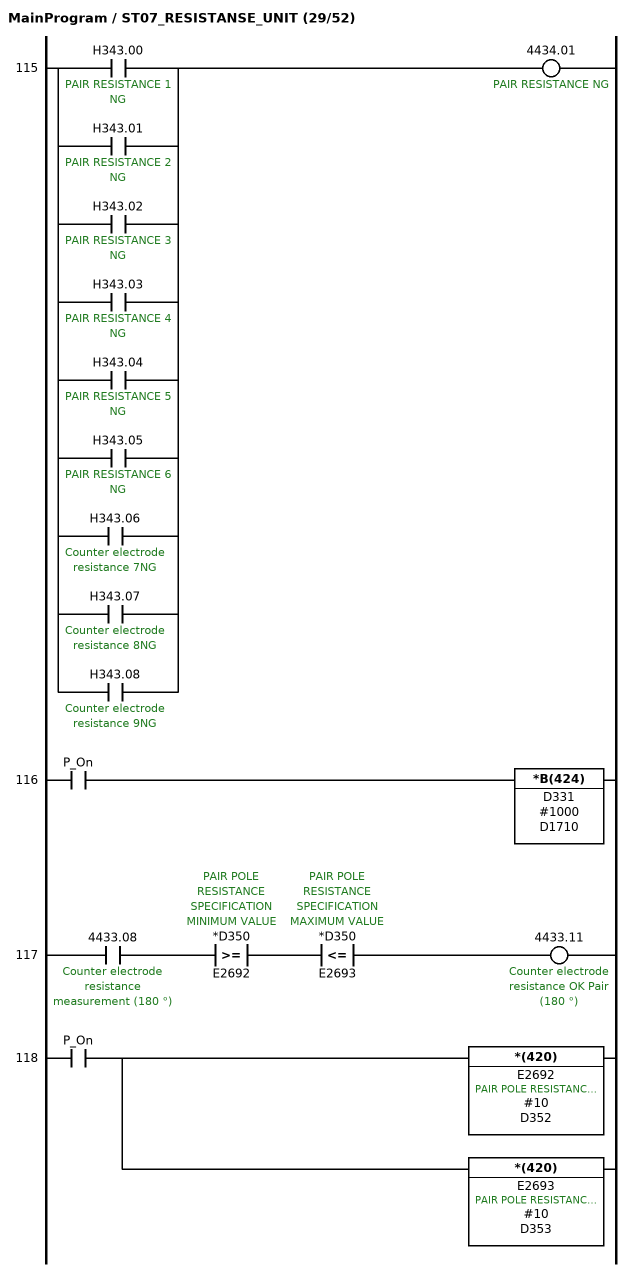
; rung 115
LD H343.00  ; PAIR RESISTANCE 1 NG
OR H343.01  ; PAIR RESISTANCE 2 NG
OR H343.02  ; PAIR RESISTANCE 3 NG
OR H343.03  ; PAIR RESISTANCE 4 NG
OR H343.04  ; PAIR RESISTANCE 5 NG
OR H343.05  ; PAIR RESISTANCE 6 NG
OR H343.06  ; Counter electrode resistance 7NG
OR H343.07  ; Counter electrode resistance 8NG
OR H343.08  ; Counter electrode resistance 9NG
OUT 4434.01  ; PAIR RESISTANCE NG
; rung 116
LD P_On
*B(424) D331 #1000 D1710
; rung 117
LD 4433.08  ; Counter electrode resistance measurement (180 °)
AND>=(325) *D350 E2692  ; PAIR POLE RESISTANCE SPECIFICATION MINIMUM VALUE
AND<=(315) *D350 E2693  ; PAIR POLE RESISTANCE SPECIFICATION MAXIMUM VALUE
OUT 4433.11  ; Counter electrode resistance OK Pair (180 °)
; rung 118
LD P_On
*(420) E2692 #10 D352  ; PAIR POLE RESISTANCE SPECIFICATION MINIMUM VALUE
*(420) E2693 #10 D353  ; PAIR POLE RESISTANCE SPECIFICATION MAXIMUM VALUE

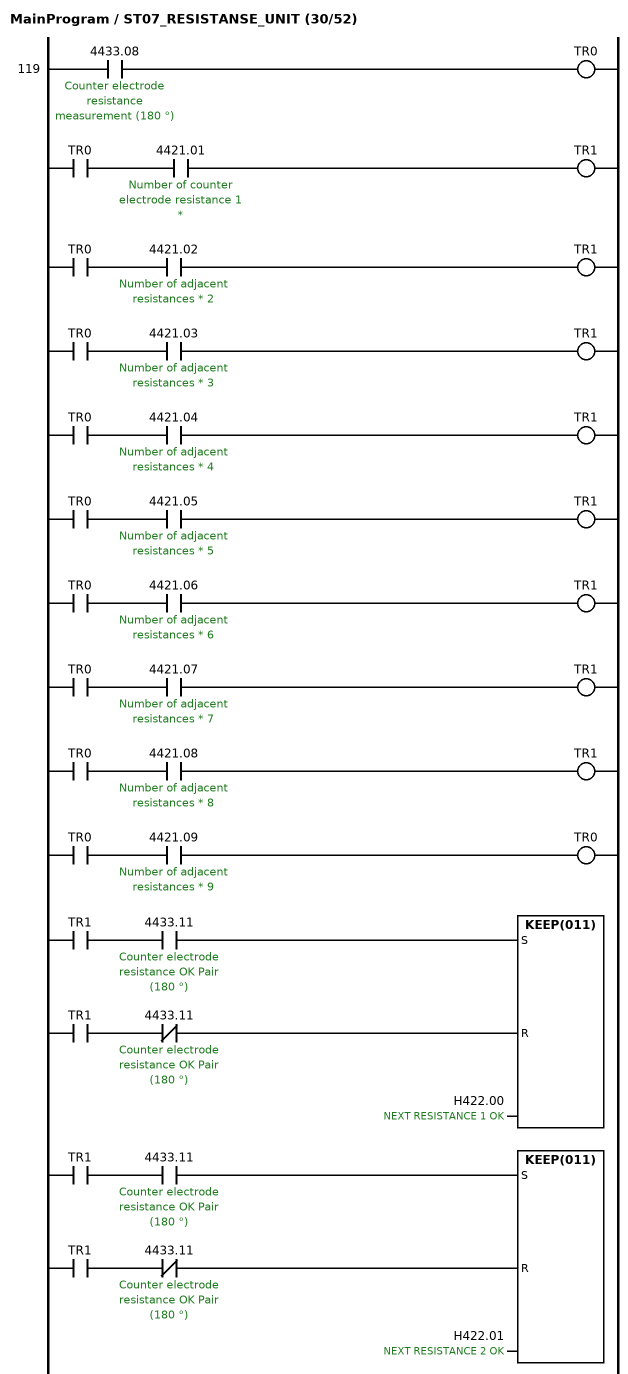

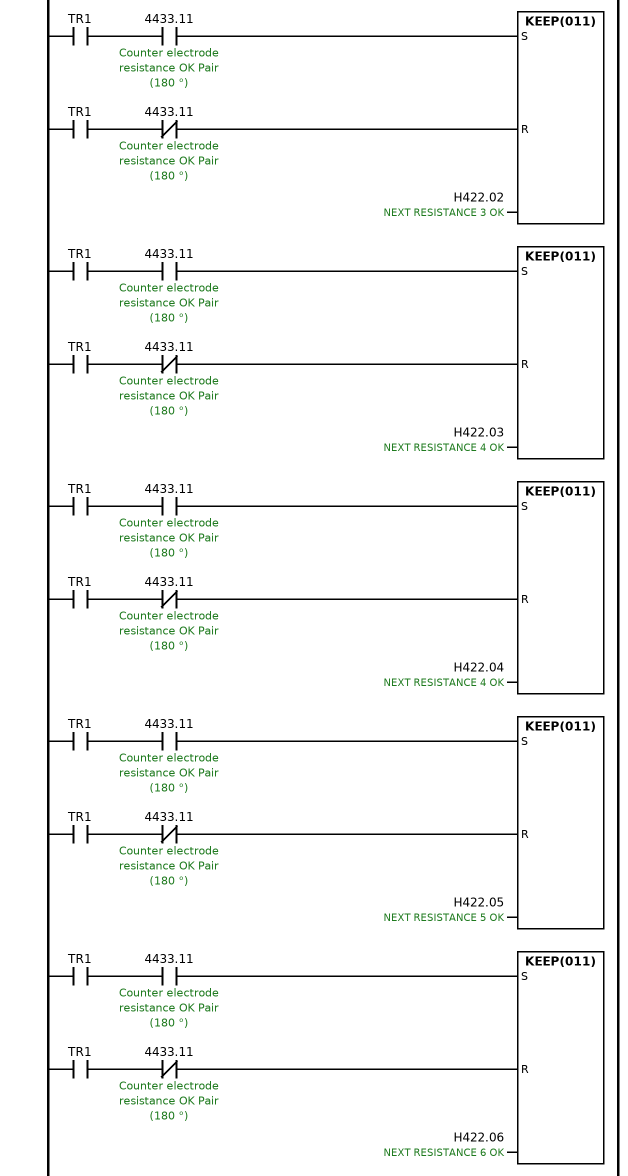

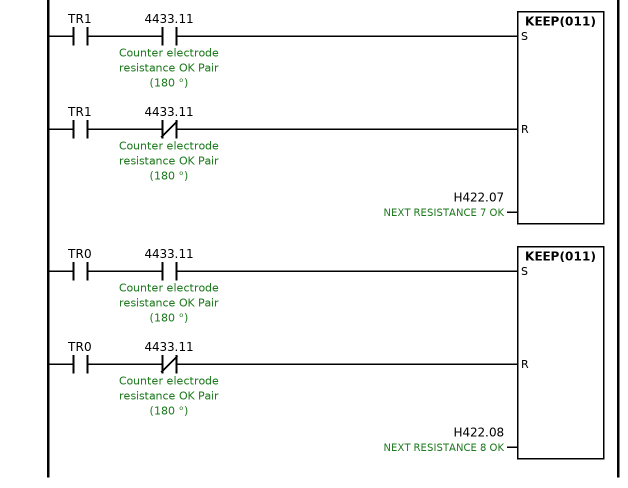
; rung 119
LD 4433.08  ; Counter electrode resistance measurement (180 °)
OUT TR0
AND 4421.01  ; Number of counter electrode resistance 1 *
OUT TR1
AND 4433.11  ; Counter electrode resistance OK Pair (180 °)
LD TR1
ANDNOT 4433.11  ; Counter electrode resistance OK Pair (180 °)
KEEP(011) H422.00  ; NEXT RESISTANCE 1 OK
LD TR0
AND 4421.02  ; Number of adjacent resistances * 2
OUT TR1
AND 4433.11  ; Counter electrode resistance OK Pair (180 °)
LD TR1
ANDNOT 4433.11  ; Counter electrode resistance OK Pair (180 °)
KEEP(011) H422.01  ; NEXT RESISTANCE 2 OK
LD TR0
AND 4421.03  ; Number of adjacent resistances * 3
OUT TR1
AND 4433.11  ; Counter electrode resistance OK Pair (180 °)
LD TR1
ANDNOT 4433.11  ; Counter electrode resistance OK Pair (180 °)
KEEP(011) H422.02  ; NEXT RESISTANCE 3 OK
LD TR0
AND 4421.04  ; Number of adjacent resistances * 4
OUT TR1
AND 4433.11  ; Counter electrode resistance OK Pair (180 °)
LD TR1
ANDNOT 4433.11  ; Counter electrode resistance OK Pair (180 °)
KEEP(011) H422.03  ; NEXT RESISTANCE 4 OK
LD TR0
AND 4421.05  ; Number of adjacent resistances * 5
OUT TR1
AND 4433.11  ; Counter electrode resistance OK Pair (180 °)
LD TR1
ANDNOT 4433.11  ; Counter electrode resistance OK Pair (180 °)
KEEP(011) H422.04  ; NEXT RESISTANCE 4 OK
LD TR0
AND 4421.06  ; Number of adjacent resistances * 6
OUT TR1
AND 4433.11  ; Counter electrode resistance OK Pair (180 °)
LD TR1
ANDNOT 4433.11  ; Counter electrode resistance OK Pair (180 °)
KEEP(011) H422.05  ; NEXT RESISTANCE 5 OK
LD TR0
AND 4421.07  ; Number of adjacent resistances * 7
OUT TR1
AND 4433.11  ; Counter electrode resistance OK Pair (180 °)
LD TR1
ANDNOT 4433.11  ; Counter electrode resistance OK Pair (180 °)
KEEP(011) H422.06  ; NEXT RESISTANCE 6 OK
LD TR0
AND 4421.08  ; Number of adjacent resistances * 8
OUT TR1
AND 4433.11  ; Counter electrode resistance OK Pair (180 °)
LD TR1
ANDNOT 4433.11  ; Counter electrode resistance OK Pair (180 °)
KEEP(011) H422.07  ; NEXT RESISTANCE 7 OK
LD TR0
AND 4421.09  ; Number of adjacent resistances * 9
OUT TR0
AND 4433.11  ; Counter electrode resistance OK Pair (180 °)
LD TR0
ANDNOT 4433.11  ; Counter electrode resistance OK Pair (180 °)
KEEP(011) H422.08  ; NEXT RESISTANCE 8 OK

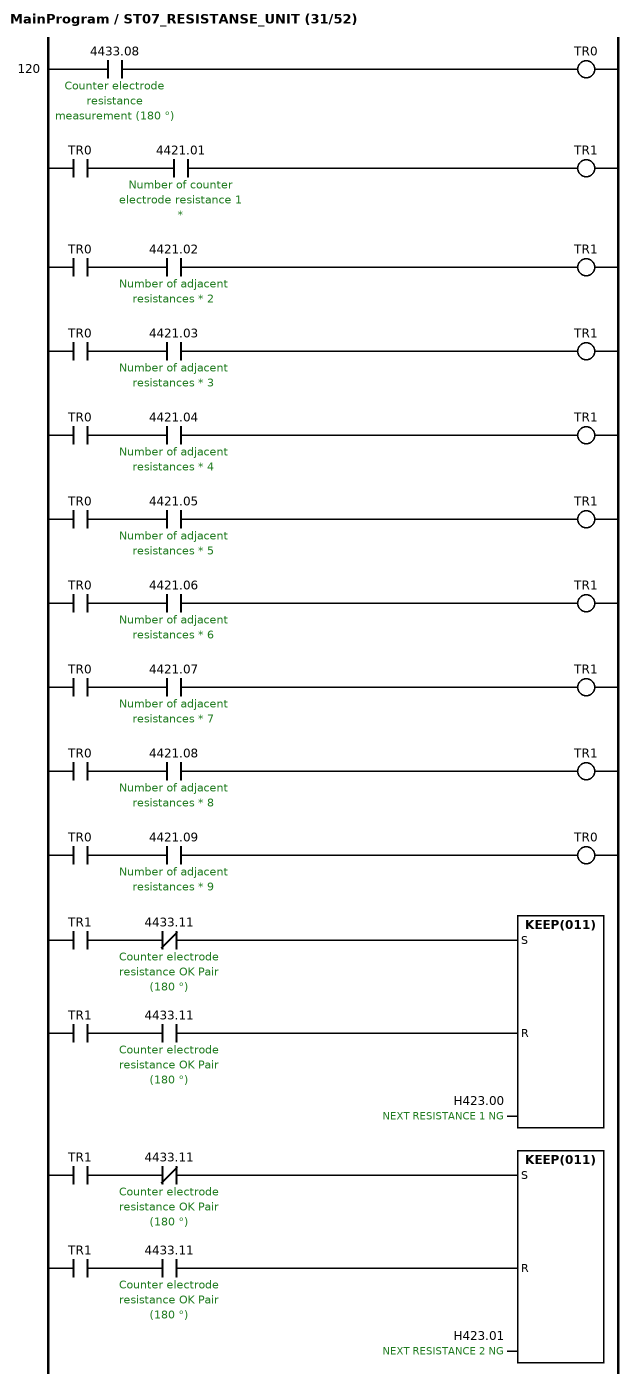

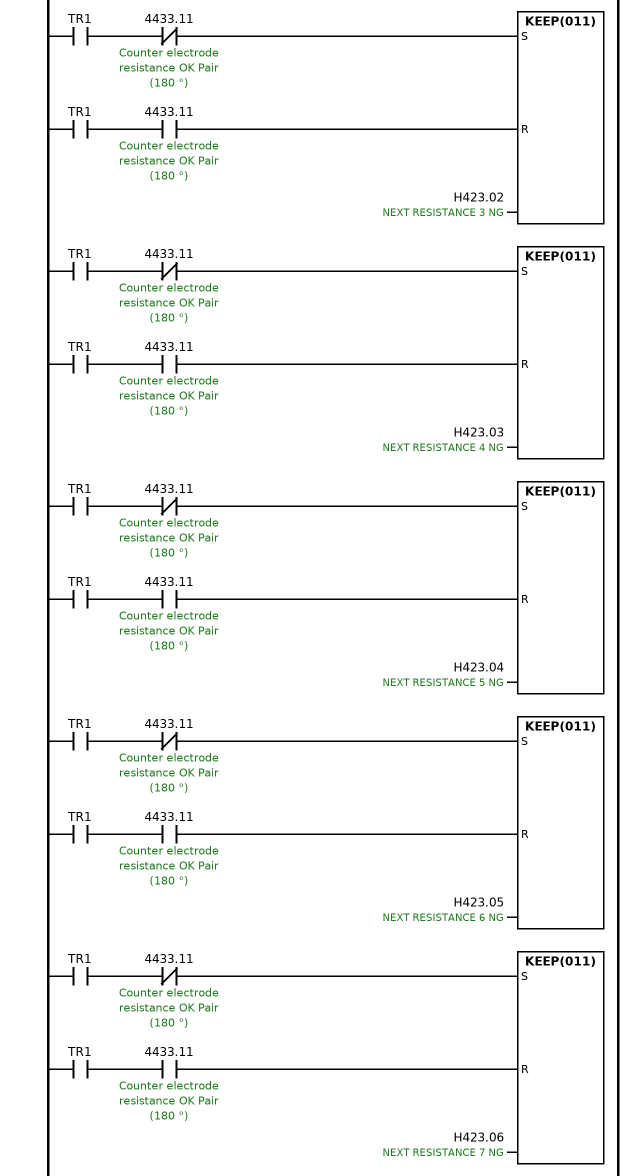

